# EPICS alarm handler configuration: alh_files/mgnt_li29_lgps.alhConfig
GROUP NULL LGPS:LI29:MG01
$ALIAS LGPS
$GUIDANCE
LI29 LGPS magnets
   Group Name: LGPS:LI29:MG01
   Summary PV:  LGPS:LI29:MG01:STATSUMY
$END

GROUP LGPS:LI29:MG01  LGPS:LI29:2
CHANNEL     LGPS:LI29:2           LGPS:LI29:2:STATMSG   -----
   $FORCEPV LGPS:LI29:2:STATMSGSV -DATL 1 0
